PROGRAM MAIN
VAR
END_VAR

Sum(3.4, 5.1);

END_PROGRAM

(* stored: Version 1.1.0.1, ProductVersion 3.1.4024.3
   POU MAIN: Id {c2cf166a-a44e-4679-95fc-9ec42efed1d2}, SpecialFunc None *)
